// TIA Portal V16 export
// export: Created 2025-05-30T16:37:07.2263402Z, ExportSetting WithDefaults, DisplayName Totally Integrated Automation Portal, DisplayVersion V16, DisplayName TIA Portal Version Control Interface, DisplayVersion V16, DisplayName TIA Portal Openness, DisplayVersion V16, DisplayName STEP 7 Professional, DisplayVersion V16, DisplayName STEP 7 Safety, DisplayVersion V16, DisplayName WinCC Advanced, DisplayVersion V16
VAR_GLOBAL   // PLC tag table "Secund. Tags"
   Aanvoerband_Tag1 AT %M100.0 : Bool;
   Aanvoerband_Tag2 AT %M100.1 : Bool;
   Trechter_Bijvullen_Haltveroorzaker AT %M100.2 : Bool;
   Safety_Automatic AT %M100.5 : Bool;
   Safety_Override AT %M100.6 : Bool;
   RUN_Automatic AT %M100.7 : Bool;
   RUN_Manual AT %M101.0 : Bool;
   Invert_Trechter_Sensor AT %M101.2 : Bool;
   WalsSensorMemory AT %M101.3 : Bool;
   Disable_Module AT %M101.4 : Bool;
   Sensor_Trechter_Delayed AT %M101.5 : Bool;
   Positive_Flank AT %M101.6 : Bool;
   ProductSensor_Flank AT %M101.7 : Bool;
   ProductSensor_Rug AT %M102.0 : Bool;
   SensorRug AT %M102.1 : Bool;
   TimeCyclusEnd AT %M102.2 : Bool;
   CounterReset AT %M102.3 : Bool;
   StartTimer AT %M102.4 : Bool;
   StopTimer AT %M102.5 : Bool;
   SaveTimervalue AT %M102.6 : Bool;
   ResetTotalProducts AT %M102.7 : Bool;
   MaintenanceNeeded AT %M103.0 : Bool;
   RetainValues AT %M112.0 : Bool;
   "Retain_1_DontTouch!" AT %M112.1 : Bool;
   Safety_Doors AT %M112.2 : Bool;
   Overname_Linked_Drive1 AT %M112.3 : Bool;
   Drive_RefuseLinkingDrive1 AT %M112.4 : Bool;
   Drive_4_Speed1_Link AT %M112.5 : Bool;
   Drive_4_Speed1_Unlink AT %M112.6 : Bool;
   SafetyOK AT %M112.7 : Bool;
   Valve2_Pulse AT %M113.0 : Bool;
END_VAR
